// TIA Portal project "babu_parkingLightQuestion" (V15)

(* hardware
DEVICE "S7-1200 station_1"  S7-1200 Station
   slot 0: "Rack_0"  S7-1200 Rack  Rack  V1.0
   slot 1: "PLC_1"  CPU 1212C DC/DC/DC  6ES7 212-1AE40-0XB0  V4.2
*)

// ===== PLC "PLC_1"  CPU 1212C DC/DC/DC =====

VAR_GLOBAL   // PLC tag table "Default tag table"
   "MEMORY BIT" AT %M0.5 : Bool;
   "MEMORY FOR EXIT DOOR" AT %M0.6 : Bool;
   "MEMORY FOR PARKING LIGHT" AT %M0.7 : Bool;
END_VAR

VAR_GLOBAL   // PLC tag table "Tag table_1"
   "S1" AT %M0.0 : Bool;
   "S2" AT %M0.1 : Bool;
   "S3" AT %M0.2 : Bool;
   "S4" AT %M0.3 : Bool;
   "S5" AT %M0.4 : Bool;
   "L1" AT %Q0.5 : Bool;
   "L2" AT %Q0.6 : Bool;
   "L3" AT %Q0.7 : Bool;
   "L4" AT %Q1.0 : Bool;
   "L5" AT %Q1.1 : Bool;
   "Exit Door Light" AT %Q1.2 : Bool;
   "Parking Area Light" AT %Q1.3 : Bool;
END_VAR

// folder: System blocks/Program resources

DATA_BLOCK "IEC_Timer_0_DB_1"   // DB2
{ S7_Optimized_Access := 'TRUE' }
AUTHOR : Simatic
FAMILY : IEC
NAME : IEC_TMR
VERSION : 1.0
// stored: InstanceOfName IEC_TIMER
"IEC_TIMER"
BEGIN
END_DATA_BLOCK

DATA_BLOCK "IEC_Timer_0_DB_2"   // DB3
{ S7_Optimized_Access := 'TRUE' }
AUTHOR : Simatic
FAMILY : IEC
NAME : IEC_TMR
VERSION : 1.0
// stored: InstanceOfName IEC_TIMER
"IEC_TIMER"
BEGIN
END_DATA_BLOCK

// folder: (top level)

ORGANIZATION_BLOCK "Main"   // OB1, LAD, ProgramCycle
TITLE = "Main Program Sweep (Cycle)"
{ S7_Optimized_Access := 'TRUE' }
VERSION : 0.1
   VAR_INPUT
      Initial_Call : Bool;   // Initial call of this OB
      Remanence : Bool;   // =True, if remanent data are available
   END_VAR
   VAR_TEMP   // added for the SCL form of the ladder/FBD networks
      _w1 : Bool;
   END_VAR
BEGIN

REGION Network 1
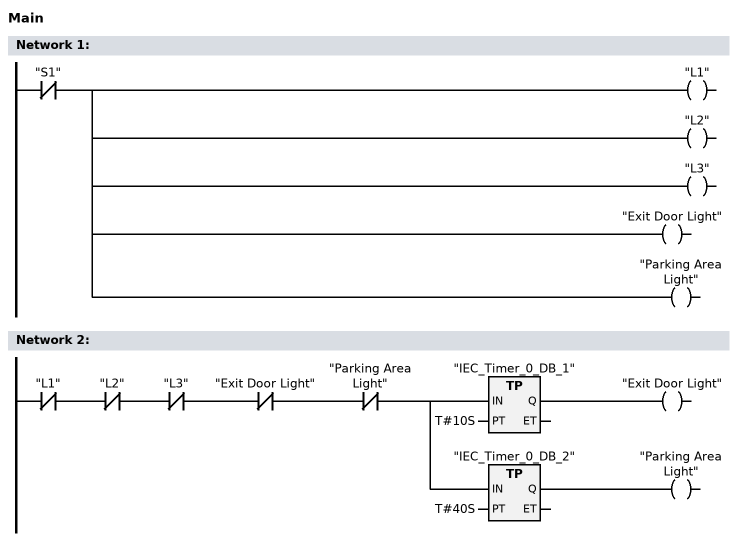
   RUNG wire#powerrail
      I_Contact( "S1" )
      wire#w1
      Coil( "L1" )
   END_RUNG
   RUNG wire#w1
      Coil( "L2" )
   END_RUNG
   RUNG wire#w1
      Coil( "L3" )
   END_RUNG
   RUNG wire#w1
      Coil( "Exit Door Light" )
   END_RUNG
   RUNG wire#w1
      Coil( "Parking Area Light" )
   END_RUNG
   // the same network as SCL:
   "L1" := NOT "S1";
   "L2" := NOT "S1";
   "L3" := NOT "S1";
   "Exit Door Light" := NOT "S1";
   "Parking Area Light" := NOT "S1";
END_REGION

REGION Network 2
   #_w1 := NOT "L1" AND NOT "L2" AND NOT "L3" AND NOT "Exit Door Light" AND NOT "Parking Area Light";
   "IEC_Timer_0_DB_1".TP(IN := #_w1, PT := T#10S);
   "Exit Door Light" := "IEC_Timer_0_DB_1".Q;
   "IEC_Timer_0_DB_2".TP(IN := #_w1, PT := T#40S);
   "Parking Area Light" := "IEC_Timer_0_DB_2".Q;
END_REGION
END_ORGANIZATION_BLOCK